FUNCTION_BLOCK FB_Timer
VAR_INPUT
	iTime	: TIME;
	execute : Bool;
END_VAR
VAR_OUTPUT
	done	: BOOL;
END_VAR
VAR
	timer	: Tc2_Standard.TON;
	state	: INT := 0;
END_VAR

IF (execute) THEN
	
	CASE state OF
	
		0:	done := FALSE;
			timer(IN:= FALSE, PT:= iTime);
			timer(IN:= TRUE, PT:= iTime);
			state := 10;
	
		10:	timer();
			IF (timer.Q) THEN
				done := TRUE;
				state :=0;
			END_IF
	END_CASE

ELSE
	state := 0;
	done := FALSE;
END_IF

END_FUNCTION_BLOCK

(* stored: Version 1.1.0.1, ProductVersion 3.1.0.25
   POU FB_Timer: Id {1b61febe-3b65-4111-88ec-89ed6a0e8231} *)
